INTERFACE I_HE_SolidAttenuatorCommands EXTENDS I_Fallible

END_INTERFACE

(* stored: Version 1.1.0.1
   Itf I_HE_SolidAttenuatorCommands: Id {967cca1c-4608-4517-b99b-1a03634089ef} *)
